PROGRAM MAIN
VAR
	axis_1:		AXIS_REF;
	FBEnable: MC_Power;
	bEnable : BOOL;
	FBAbsolute: MC_MoveAbsolute;
	bAbsolute : BOOL;
	
	fb_absolute_Example    : FB_Absolute_Example;
	Axis1: AXIS_REF;
	fPosition1:		 LREAL;
	fPosition2:		 LREAL;
	fPosition3		:LREAL;
	tDelay: 		 TIME;
	fVelocity:		 LREAL;
	bError:			 BOOL;
	sStatus:		 STRING;
	
	bBool			:BOOL;
	bBool1: INT;
	fb_Reset: MC_Reset;
	
	
   
    bBoool	:		BOOL;
	position	:	LREAL;
	mode		:	BOOL;
	options		:ST_SetPositionOptions;
	fb_SetPosition: MC_SetPosition;
END_VAR



fb_absolute_Example(
	bEnable:=bEnable , 
	fPosition1:= fPosition1, 
	fPosition2:=fPosition2 , 
	fPosition3:= fPosition3, 
	tDelay:= tDelay, 
	fVelocity:= fVelocity, 
	bError=>bError , 
	sStatus=>sStatus , 
	Axis:=axis_1 );

END_PROGRAM

(* stored: Version 1.1.0.1, ProductVersion 3.1.4024.12
   POU MAIN: Id {785e37b4-1199-4605-b604-bae944d0423f}, SpecialFunc None *)
